// Mitsubishi GX Works2 project: 32 ramp on off   PLC: Q02/Q02H

PROGRAM MAIN
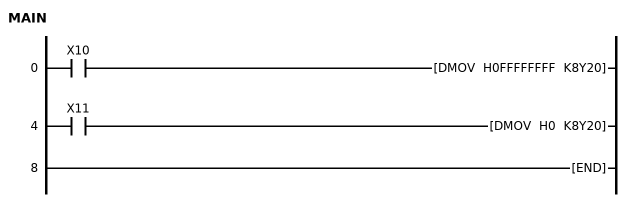
0     LD      X10
      DMOV    H0FFFFFFFF K8Y20
4     LD      X11
      DMOV    H0 K8Y20
8     END
END_PROGRAM
